(*
SPDX-FileCopyrightText: © 2026 Oleksandr Tiutyk <trofimich@gmail.com>
SPDX-License-Identifier: MIT
License: https://opensource.org/license/mit
*)

(*!
<summary>Exposes diagnostics for a rejected filesystem path.</summary>
<description>
Reports caller-detected path errors using the GeneralException lifetime and throw rules. The path is borrowed
during the call; errorMessage is copied by value.
</description>
*)
INTERFACE IInvalidPathException EXTENDS TOF_Core.IGeneralException

(*!
<summary>Raises an exception describing the rejected path and its reason.</summary>
<description>
Borrows path read-only for this call and copies errorMessage by value, limited to 255 characters. Retains
formatted diagnostic text, not the input reference. The caller detects the invalid path; this method does not
validate it.
</description>
*)
METHOD Throw
VAR_INPUT
	sourceNamespaceName : STRING;
	sourceClassName : STRING;
	sourcePOUName : STRING;
	sourcePosition : STRING;
END_VAR
VAR_IN_OUT CONSTANT
	path : STRING(255);
END_VAR
VAR_INPUT
	errorMessage : WSTRING(255);
END_VAR
END_METHOD

END_INTERFACE

(* stored: Version 1.1.0.1
   Itf IInvalidPathException: Id {4fabf056-d31d-48b6-bc73-597bed22690b}
   Method Throw: Id {3aecdf47-2204-47ee-b3e1-2f24c9af88aa} *)
